// SIMATIC S7-200 project (STEP 7-Micro/WIN), CPU 224XP REL 02.01

SYMBOL_TABLE USUARIO1
P_MARCHA         I0.0
P_PARO           I0.1
TERMICO          I0.2
M_BOMBA_ACEITE   Q0.0
LED_MARCHA       Q0.1
MP_LINEA         Q0.2
MP_ESTRELLA      Q0.3
MP_TRIANGULO     Q0.4
LED_PARO         Q0.5
LED_AVERIA       Q0.6
SIMULACION_FALLO I0.3
END_SYMBOL_TABLE

ORGANIZATION_BLOCK PRINCIPAL:OB1
TITLE=COMENTARIOS DEL PROGRAMA
BEGIN
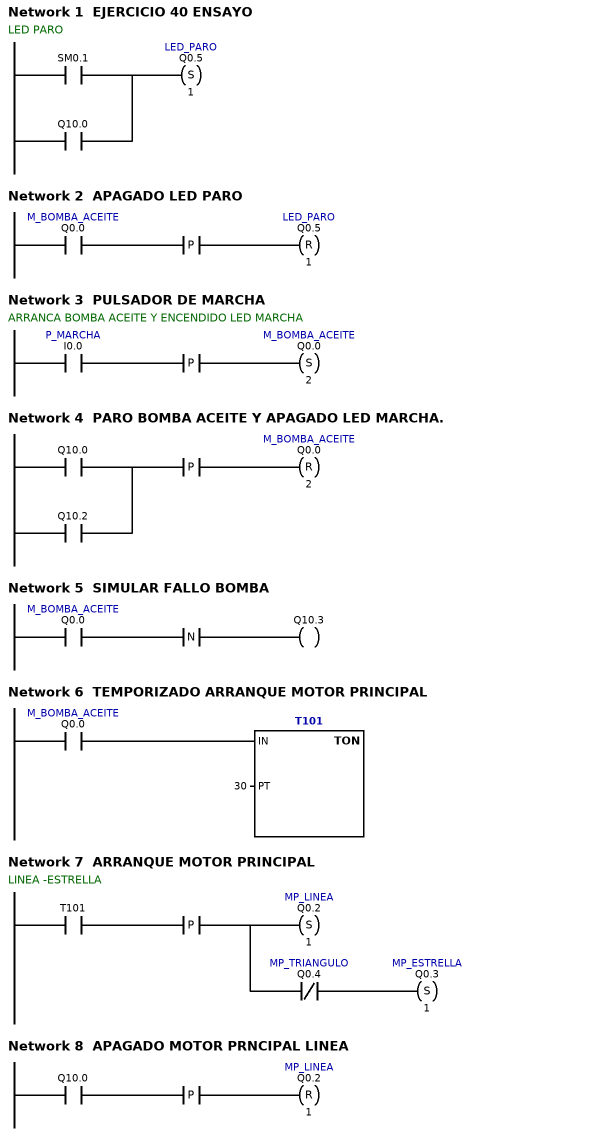
Network 1 // EJERCICIO 40 ENSAYO
// LED PARO
LD     SM0.1
O      Q10.0
S      LED_PARO:Q0.5, 1
Network 2 // APAGADO LED PARO
LD     M_BOMBA_ACEITE:Q0.0
EU
R      LED_PARO:Q0.5, 1
Network 3 // PULSADOR DE MARCHA
// ARRANCA BOMBA ACEITE Y ENCENDIDO LED MARCHA
LD     P_MARCHA:I0.0
EU
S      M_BOMBA_ACEITE:Q0.0, 2
Network 4 // PARO BOMBA ACEITE Y APAGADO LED MARCHA.
LD     Q10.0
O      Q10.2
EU
R      M_BOMBA_ACEITE:Q0.0, 2
Network 5 // SIMULAR FALLO BOMBA
LD     M_BOMBA_ACEITE:Q0.0
ED
=      Q10.3
Network 6 // TEMPORIZADO ARRANQUE MOTOR PRINCIPAL
LD     M_BOMBA_ACEITE:Q0.0
TON    T101, 30
Network 7 // ARRANQUE MOTOR PRINCIPAL
// LINEA -ESTRELLA
LD     T101
EU
S      MP_LINEA:Q0.2, 1
AN     MP_TRIANGULO:Q0.4
S      MP_ESTRELLA:Q0.3, 1
Network 8 // APAGADO MOTOR PRNCIPAL LINEA
LD     Q10.0
EU
R      MP_LINEA:Q0.2, 1
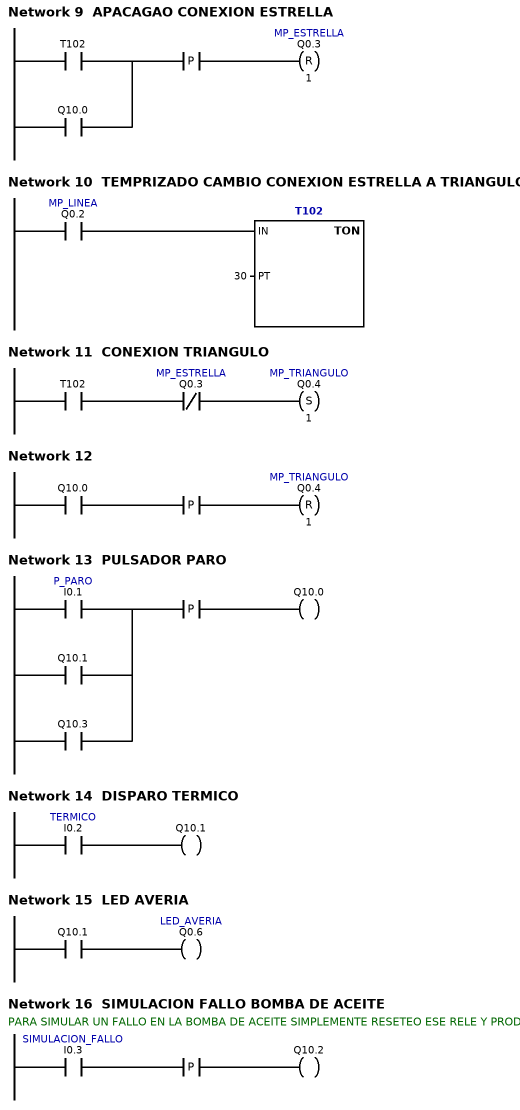
Network 9 // APACAGAO CONEXION ESTRELLA
LD     T102
O      Q10.0
EU
R      MP_ESTRELLA:Q0.3, 1
Network 10 // TEMPRIZADO CAMBIO CONEXION ESTRELLA A TRIANGULO
LD     MP_LINEA:Q0.2
TON    T102, 30
Network 11 // CONEXION TRIANGULO
LD     T102
AN     MP_ESTRELLA:Q0.3
S      MP_TRIANGULO:Q0.4, 1
Network 12
LD     Q10.0
EU
R      MP_TRIANGULO:Q0.4, 1
Network 13 // PULSADOR PARO
LD     P_PARO:I0.1
O      Q10.1
O      Q10.3
EU
=      Q10.0
Network 14 // DISPARO TERMICO
LD     TERMICO:I0.2
=      Q10.1
Network 15 // LED AVERIA
LD     Q10.1
=      LED_AVERIA:Q0.6
Network 16 // SIMULACION FALLO BOMBA DE ACEITE
// PARA SIMULAR UN FALLO EN LA BOMBA DE ACEITE SIMPLEMENTE RESETEO ESE RELE Y PRODUCIRA LA PARADA MEDIANTE UN IMPULSO AL RESET DE MOTOR PRINCIPAL.
LD     SIMULACION_FALLO:I0.3
EU
=      Q10.2
END_ORGANIZATION_BLOCK
